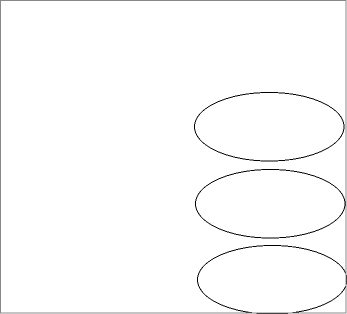
VISUALIZATION Visualization  // 347x314
    Ellipse (194,92 150x69), colour toggle: MAIN.bRed
    Ellipse (195,169 150x69), colour toggle: MAIN.bAmber
    Ellipse (197,245 150x69), colour toggle: MAIN.bGreen
END_VISUALIZATION

(* stored: Version 1.1.0.1, ProductVersion 3.1.4024.16
   Visu Visualization: Id {9e4652b4-c52c-4815-b926-ee532e6ae218} *)
